// TIA Portal V19 export
TYPE "TetraPakV70_10_Params"
TITLE = TPV70_10_Params
// DEVICEID : 10
//  VENDOR : IFM on behalf of Tetra Pak
//  DATE: 27.12.2023 
// 
//  Comment : TPV70_10_Params
   STRUCT
      StandardStructure : Struct
         Header : Struct
            NumberParameter : Int := 20;   // Number of device parameters (Device Identification + Device Parameter)
            AdressParamDownLoad : Int := 20;   // Start adress for ParamDownload signals in this struct
            AdressDeviceIndent : Int := 44;   // Start adress for Device Identification Parameters in this struct
            AdressApplicSpez : Int := 536;   // Start adress ApplicationSpezificTag
            AdressDeviceParam : Int := 782;   // Start adress for Device Parameters in this Area
            AdressKommando : Int := 1004;   // Start adress for Device Commandos
            NumberCommandos : Int := 5;   // Number of Commandos of the device
            Spare01 : Int;   // spare
            Spare02 : Int;   // spare
            Spare03 : Int;   // spare
         END_STRUCT;
         Paramdownload : Struct
            ParamDownLoadStart : Struct   // Parameter Download Start (Only if master and device are V1.1)
               BlockStat : DWord;   // function block status
               IOLStat : DWord;   // IO-Link Status
            END_STRUCT;
            ParamDownLoadEnd : Struct   // Parameter Download End (Only if master and device are V1.1)
               BlockStat : DWord;   // function block status
               IOLStat : DWord;   // IO-Link Status
            END_STRUCT;
            ParamDownLoadStore : Struct   // Parameter Download Store (Only if master and device are V1.1)
               BlockStat : DWord;   // function block status
               IOLStat : DWord;   // IO-Link Status
            END_STRUCT;
         END_STRUCT;
         DeviceIndentification : Struct   // device indentification parameter
            V_VendorName : Struct   // Vendor Name
               Text : String[64];
               Index : Int := 16;   // parameter index
               Subindex : Int;   // parameter subindex
               Length : Int := 10;   // parameter length in BYTE for writing
               BlockStat : DWord;   // function block status
               IOLStat : DWord;   // IO-Link Status
               RelRead : Bool := TRUE;   // reading release
               RelWrite : Bool;   // writing release
            END_STRUCT;
            V_ProductName : Struct   // Product Name
               Text : String[64];
               Index : Int := 18;   // parameter index
               Subindex : Int;   // parameter subindex
               Length : Int := 20;   // parameter length in BYTE for writing
               BlockStat : DWord;   // function block status
               IOLStat : DWord;   // IO-Link Status
               RelRead : Bool := TRUE;   // reading release
               RelWrite : Bool;   // writing release
            END_STRUCT;
            V_ProductID : Struct   // Product ID
               Text : String[64];
               Index : Int := 19;   // parameter index
               Subindex : Int;   // parameter subindex
               Length : Int := 20;   // parameter length in BYTE for writing
               BlockStat : DWord;   // function block status
               IOLStat : DWord;   // IO-Link Status
               RelRead : Bool := TRUE;   // reading release
               RelWrite : Bool;   // writing release
            END_STRUCT;
            V_ProductText : Struct   // Product Text
               Text : String[64];
               Index : Int := 20;   // parameter index
               Subindex : Int;   // parameter subindex
               Length : Int := 31;   // parameter length in BYTE for writing
               BlockStat : DWord;   // function block status
               IOLStat : DWord;   // IO-Link Status
               RelRead : Bool := TRUE;   // reading release
               RelWrite : Bool;   // writing release
            END_STRUCT;
            V_HardwareRevision : Struct   // Hardware Version
               Text : String[64];
               Index : Int := 22;   // parameter index
               Subindex : Int;   // parameter subindex
               Length : Int := 2;   // parameter length in BYTE for writing
               BlockStat : DWord;   // function block status
               IOLStat : DWord;   // IO-Link Status
               RelRead : Bool := TRUE;   // reading release
               RelWrite : Bool;   // writing release
            END_STRUCT;
            V_FirmwareRevision : Struct   // Firmware Version
               Text : String[64];
               Index : Int := 23;   // parameter index
               Subindex : Int;   // parameter subindex
               Length : Int := 16;   // parameter length in BYTE for writing
               BlockStat : DWord;   // function block status
               IOLStat : DWord;   // IO-Link Status
               RelRead : Bool := TRUE;   // reading release
               RelWrite : Bool;   // writing release
            END_STRUCT;
         END_STRUCT;
         ApplicationSpecificTag : Struct   // AppliciationSpecificTag
            V_ApplicationSpecificTa : Struct   // Application Specific Tag
               Text : String[64];
               Index : Int := 24;   // parameter index
               Subindex : Int;   // parameter subindex
               Length : Int := 32;   // parameter length in BYTE for writing
               BlockStat : DWord;   // function block status
               IOLStat : DWord;   // IO-Link Status
               RelRead : Bool := TRUE;   // reading release
               RelWrite : Bool := TRUE;   // writing release
            END_STRUCT;
            V_FunctionTag : Struct   // Function Tag
               Text : String[64];
               Index : Int := 25;   // parameter index
               Subindex : Int;   // parameter subindex
               Length : Int := 32;   // parameter length in BYTE for writing
               BlockStat : DWord;   // function block status
               IOLStat : DWord;   // IO-Link Status
               RelRead : Bool := TRUE;   // reading release
               RelWrite : Bool := TRUE;   // writing release
            END_STRUCT;
            V_LocationTag : Struct   // Location Tag
               Text : String[64];
               Index : Int := 26;   // parameter index
               Subindex : Int;   // parameter subindex
               Length : Int := 32;   // parameter length in BYTE for writing
               BlockStat : DWord;   // function block status
               IOLStat : DWord;   // IO-Link Status
               RelRead : Bool := TRUE;   // reading release
               RelWrite : Bool := TRUE;   // writing release
            END_STRUCT;
         END_STRUCT;
         DeviceParameters : Struct   // Device Parameters
            Parameter_01 : Struct   // V_DeviceAccessLocks > Device Access Locks
               Value : Struct   // Parameter Value (must be always 4 Byte)
                  V_DeviceAccessLocks : Int;
                  Byte02 : Byte;
                  Byte03 : Byte;
               END_STRUCT;
               Index : Int := 12;   // parameter index
               Subindex : Int;   // parameter subindex
               Length : Int := 2;   // parameter length in BYTE for writing
               BlockStat : DWord;   // function block status
               IOLStat : DWord;   // IO-Link Status
               RelRead : Bool := TRUE;   // reading release
               RelWrite : Bool := TRUE;   // writing release
            END_STRUCT;
            Parameter_02 : Struct   // The stroke durations per solenoid valve SV1 (energizing direction)
               Value : Struct   // Parameter Value (must be always 4 Byte)
                  StrokeDurationSV1EN : DInt;   // ms
               END_STRUCT;
               Index : Int := 85;   // parameter index
               Subindex : Int := 1;   // parameter subindex
               Length : Int := 4;   // parameter length in BYTE for writing
               BlockStat : DWord;   // function block status
               IOLStat : DWord;   // IO-Link Status
               RelRead : Bool := TRUE;   // reading release
               RelWrite : Bool;   // writing release
            END_STRUCT;
            Parameter_03 : Struct   // The stroke durations per solenoid valve SV2 (energizing direction)
               Value : Struct   // Parameter Value (must be always 4 Byte)
                  StrokeDurationSV2EN : DInt;   // ms
               END_STRUCT;
               Index : Int := 85;   // parameter index
               Subindex : Int := 2;   // parameter subindex
               Length : Int := 4;   // parameter length in BYTE for writing
               BlockStat : DWord;   // function block status
               IOLStat : DWord;   // IO-Link Status
               RelRead : Bool := TRUE;   // reading release
               RelWrite : Bool;   // writing release
            END_STRUCT;
            Parameter_04 : Struct   // The stroke durations per solenoid valve SV3(energizing direction)
               Value : Struct   // Parameter Value (must be always 4 Byte)
                  StrokeDurationSV3EN : DInt;   // ms
               END_STRUCT;
               Index : Int := 85;   // parameter index
               Subindex : Int := 3;   // parameter subindex
               Length : Int := 4;   // parameter length in BYTE for writing
               BlockStat : DWord;   // function block status
               IOLStat : DWord;   // IO-Link Status
               RelRead : Bool := TRUE;   // reading release
               RelWrite : Bool;   // writing release
            END_STRUCT;
            Parameter_05 : Struct   // The setup stroke durations pr solenoid valve SV1(de-energizing direction)
               Value : Struct   // Parameter Value (must be always 4 Byte)
                  StrokeDurationSV1DEEN : DInt;   // ms
               END_STRUCT;
               Index : Int := 86;   // parameter index
               Subindex : Int := 1;   // parameter subindex
               Length : Int := 4;   // parameter length in BYTE for writing
               BlockStat : DWord;   // function block status
               IOLStat : DWord;   // IO-Link Status
               RelRead : Bool := TRUE;   // reading release
               RelWrite : Bool;   // writing release
            END_STRUCT;
            Parameter_06 : Struct   // The setup stroke durations pr solenoid valve SV2(de-energizing direction)
               Value : Struct   // Parameter Value (must be always 4 Byte)
                  StrokeDurationSV2DEEN : DInt;   // ms
               END_STRUCT;
               Index : Int := 86;   // parameter index
               Subindex : Int := 2;   // parameter subindex
               Length : Int := 4;   // parameter length in BYTE for writing
               BlockStat : DWord;   // function block status
               IOLStat : DWord;   // IO-Link Status
               RelRead : Bool := TRUE;   // reading release
               RelWrite : Bool;   // writing release
            END_STRUCT;
            Parameter_07 : Struct   // The setup stroke durations pr solenoid valve SV3(de-energizing direction)
               Value : Struct   // Parameter Value (must be always 4 Byte)
                  StrokeDurationSV3DEEN : DInt;   // ms
               END_STRUCT;
               Index : Int := 86;   // parameter index
               Subindex : Int := 3;   // parameter subindex
               Length : Int := 4;   // parameter length in BYTE for writing
               BlockStat : DWord;   // function block status
               IOLStat : DWord;   // IO-Link Status
               RelRead : Bool := TRUE;   // reading release
               RelWrite : Bool;   // writing release
            END_STRUCT;
            Parameter_08 : Struct   // Number of solenoid valve activations SV1
               Value : Struct   // Parameter Value (must be always 4 Byte)
                  SV1Activations : DInt;
               END_STRUCT;
               Index : Int := 83;   // parameter index
               Subindex : Int := 1;   // parameter subindex
               Length : Int := 4;   // parameter length in BYTE for writing
               BlockStat : DWord;   // function block status
               IOLStat : DWord;   // IO-Link Status
               RelRead : Bool := TRUE;   // reading release
               RelWrite : Bool;   // writing release
            END_STRUCT;
            Parameter_09 : Struct   // Number of solenoid valve activations SV2
               Value : Struct   // Parameter Value (must be always 4 Byte)
                  SV2Activations : DInt;
               END_STRUCT;
               Index : Int := 83;   // parameter index
               Subindex : Int := 2;   // parameter subindex
               Length : Int := 4;   // parameter length in BYTE for writing
               BlockStat : DWord;   // function block status
               IOLStat : DWord;   // IO-Link Status
               RelRead : Bool := TRUE;   // reading release
               RelWrite : Bool;   // writing release
            END_STRUCT;
            Parameter_10 : Struct   // Number of solenoid valve activations SV3
               Value : Struct   // Parameter Value (must be always 4 Byte)
                  SV3Activations : DInt;
               END_STRUCT;
               Index : Int := 83;   // parameter index
               Subindex : Int := 3;   // parameter subindex
               Length : Int := 2;   // parameter length in BYTE for writing
               BlockStat : DWord;   // function block status
               IOLStat : DWord;   // IO-Link Status
               RelRead : Bool := TRUE;   // reading release
               RelWrite : Bool;   // writing release
            END_STRUCT;
            Parameter_11 : Struct   // Logging information runtime
               Value : Struct   // Parameter Value (must be always 4 Byte)
                  RunTime : DInt;
               END_STRUCT;
               Index : Int := 80;   // parameter index
               Subindex : Int := 2;   // parameter subindex
               Length : Int := 4;   // parameter length in BYTE for writing
               BlockStat : DWord;   // function block status
               IOLStat : DWord;   // IO-Link Status
               RelRead : Bool := TRUE;   // reading release
               RelWrite : Bool;   // writing release
            END_STRUCT;
         END_STRUCT;
         Commando : Struct   // Commandos
            Commando_00 : Struct   // Restore Factory Settings
               Value : Byte := BYTE#16#82;   // 130
               Index : Int := 2;   // parameter index
               Subindex : Int;   // parameter subindex
               Length : Int := 1;   // parameter length in BYTE for writing
               BlockStat : DWord;   // function block status
               IOLStat : DWord;   // IO-Link Status
            END_STRUCT;
            Commando_01 : Struct   // Start Auto Setup
               Value : Byte := BYTE#16#D0;   // 208
               Index : Int := 2;   // parameter index
               Subindex : Int;   // parameter subindex
               Length : Int := 1;   // parameter length in BYTE for writing
               BlockStat : DWord;   // function block status
               IOLStat : DWord;   // IO-Link Status
            END_STRUCT;
            Commando_02 : Struct   // Setup Reset
               Value : Byte := BYTE#16#D1;   // 209
               Index : Int := 2;   // parameter index
               Subindex : Int;   // parameter subindex
               Length : Int := 1;   // parameter length in BYTE for writing
               BlockStat : DWord;   // function block status
               IOLStat : DWord;   // IO-Link Status
            END_STRUCT;
            Commando_03 : Struct   // Parameter Reset
               Value : Byte := BYTE#16#D2;   // 210
               Index : Int := 2;   // parameter index
               Subindex : Int;   // parameter subindex
               Length : Int := 1;   // parameter length in BYTE for writing
               BlockStat : DWord;   // function block status
               IOLStat : DWord;   // IO-Link Status
            END_STRUCT;
            Commando_04 : Struct   // Diagnostic Reset
               Value : Byte := BYTE#16#D3;   // 211
               Index : Int := 2;   // parameter index
               Subindex : Int;   // parameter subindex
               Length : Int := 1;   // parameter length in BYTE for writing
               BlockStat : DWord;   // function block status
               IOLStat : DWord;   // IO-Link Status
            END_STRUCT;
         END_STRUCT;
      END_STRUCT;
   END_STRUCT;
END_TYPE
